{attribute addProperty BoxType "AX2000-B110-0000"}
{attribute addProperty Id "Velocity_demand_valueAT %Q*DINT3240Control_wordAT %Q*UINT1620"}
{attribute addProperty CRC "968198527"}
{attribute addProperty SizeInBites "48"}
{attribute addProperty SizeInBytes "6"}
TYPE Outputs_39B5897F :
STRUCT
	{attribute addProperty Name "Velocity_demand_value"}
	Velocity_demand_value AT %Q* : DINT;
	{attribute addProperty Name "Control_word"}
	Control_word AT %Q* : UINT;
END_STRUCT
END_TYPE

(* stored: Version 1.2.0.0, ProductVersion 3.1.4024.9
   DUT Outputs_39B5897F: Id {286c9d50-8afc-45e8-8a1e-c529a07908bd} *)
